// TIA Portal V20 export
FUNCTION_BLOCK "LER_Actuator"   // FB30, LAD
// stored: Access Published, MemoryReserve 100, Namespace Cylinder, SetENOAutomatically false
   VAR_INPUT
      Status : "LAF_typeUnitStatus";
      HMI : Bool;
      Process : Bool;
      int1 { ExternalAccessible := 'False'; ExternalVisible := 'False'; ExternalWritable := 'False'} : Bool := true;
      int2 { ExternalAccessible := 'False'; ExternalVisible := 'False'; ExternalWritable := 'False'} : Bool := true;
      int3 { ExternalAccessible := 'False'; ExternalVisible := 'False'; ExternalWritable := 'False'} : Bool := true;
      int4 { ExternalAccessible := 'False'; ExternalVisible := 'False'; ExternalWritable := 'False'} : Bool := true;
      int5 { ExternalAccessible := 'False'; ExternalVisible := 'False'; ExternalWritable := 'False'} : Bool := true;
      int6 { ExternalAccessible := 'False'; ExternalVisible := 'False'; ExternalWritable := 'False'} : Bool := true;
      int7 { ExternalAccessible := 'False'; ExternalVisible := 'False'; ExternalWritable := 'False'} : Bool := true;
      int8 { ExternalAccessible := 'False'; ExternalVisible := 'False'; ExternalWritable := 'False'} : Bool := true;
      int9 { ExternalAccessible := 'False'; ExternalVisible := 'False'; ExternalWritable := 'False'} : Bool := true;
      int10 { ExternalAccessible := 'False'; ExternalVisible := 'False'; ExternalWritable := 'False'} : Bool := true;
      Bypass : Bool := true;
   END_VAR
   VAR_OUTPUT
      Moveing_INT : Bool;
   END_VAR
   VAR_IN_OUT
      intOut : Array[0..9] of Bool;
   END_VAR
   VAR
      condition_moveing : Bool;
      NotCondition_moveing { ExternalVisible := 'False'} : Bool;
   END_VAR
BEGIN

REGION Network 2 (SCL)


   IF (#int1 AND #int2 AND #int3 AND #int4 AND #int5 AND #int6 AND #int7 AND #int8 AND #int9 AND #int10 )OR #Bypass THEN

           #condition_moveing := TRUE;
           #NotCondition_moveing := FALSE;
           IF #HMI OR #Process THEN

                   #intOut[0] := FALSE;
                   #intOut[1] := FALSE;
                   #intOut[2] := FALSE;
                   #intOut[3] := FALSE;
                   #intOut[4] := FALSE;
                   #intOut[5] := FALSE;
                   #intOut[6] := FALSE;
                   #intOut[7] := FALSE;
                   #intOut[8] := FALSE;
                   #intOut[9] := FALSE;

           END_IF;
     ELSE
          #condition_moveing := FALSE;
          #NotCondition_moveing := TRUE;
          IF #HMI OR #Process THEN
              IF NOT #int1 THEN
                   #intOut[0] := TRUE;
               ELSE
                   #intOut[0] := FALSE;
               END_IF;
               IF NOT #int2 THEN
                   #intOut[1] := TRUE;
               ELSE
                   #intOut[1] := FALSE;
               END_IF;
               IF NOT #int3 THEN
                   #intOut[2] := TRUE;
               ELSE
                   #intOut[2] := FALSE;
               END_IF;
               IF NOT #int4 THEN
                   #intOut[3] := TRUE;
               ELSE
                   #intOut[3] := FALSE;
               END_IF;
               IF NOT #int5 THEN
                   #intOut[4] := TRUE;
               ELSE
                   #intOut[4] := FALSE;
               END_IF;
               IF NOT #int6 THEN
                   #intOut[5] := TRUE;
               ELSE
                   #intOut[5] := FALSE;
               END_IF;
               IF NOT #int7 THEN
                   #intOut[6] := TRUE;
               ELSE
                   #intOut[6] := FALSE;
               END_IF;
               IF NOT #int8 THEN
                   #intOut[7] := TRUE;
               ELSE
                   #intOut[7] := FALSE;
               END_IF;
               IF NOT #int9 THEN
                   #intOut[8] := TRUE;
               ELSE
                   #intOut[8] := FALSE;
               END_IF;
               IF NOT #int10 THEN
                   #intOut[9] := TRUE;
               ELSE
                   #intOut[9] := FALSE;
               END_IF;


         END_IF;

     END_IF;

   #Moveing_INT := #condition_moveing;
END_REGION
END_FUNCTION_BLOCK
